// TIA Portal V20 export
DATA_BLOCK "InstCycleTimerDataset3"   // DB178
TITLE = Instanz CycleTimerDataset2 / Instance CycleTimerDataset2
{ DB_Accessible_From_OPC_UA := 'FALSE' }
AUTHOR : SICAR
FAMILY : ProdData
// Instanz DB / Instance DB
// stored: DBAccessibleFromOPCUA false, InstanceOfName LSicar_ProdDataCycleTimer, InstanceOfType FB
"LSicar_ProdDataCycleTimer"
   // VAR_INPUT
   //    numberConfigDataSets { ExternalAccessible := 'False'; ExternalVisible := 'False'; ExternalWritable := 'False'} : Int;
   //    dataSetNumber { ExternalAccessible := 'False'; ExternalVisible := 'False'; ExternalWritable := 'False'} : UInt;
   //    pulse100ms { ExternalAccessible := 'False'; ExternalVisible := 'False'; ExternalWritable := 'False'} : Bool;
   // END_VAR
   // VAR_IN_OUT
   //    numberOfDataSets : "LSicar_typeNumberOfDataSets";
   //    dataSet : "LSicar_typeCycleTimer";
   // END_VAR
   // VAR
   //    statCycleTimer { ExternalAccessible := 'False'; ExternalVisible := 'False'; ExternalWritable := 'False'} : Array[0..20] of "LSicar_typeCycleTimerStruct";
   //    statRisEdgeResetAllExt { ExternalAccessible := 'False'; ExternalVisible := 'False'; ExternalWritable := 'False'} : Bool;
   //    statPosPulseResetAllExt { ExternalAccessible := 'False'; ExternalVisible := 'False'; ExternalWritable := 'False'} : Bool;
   //    statRisEdgeResetAll { ExternalAccessible := 'False'; ExternalVisible := 'False'; ExternalWritable := 'False'} : Bool;
   //    statPosPulseResetAll { ExternalAccessible := 'False'; ExternalVisible := 'False'; ExternalWritable := 'False'} : Bool;
   // END_VAR
BEGIN
END_DATA_BLOCK
